// TwinCAT 3 PLC project Untitled2
// Title: Projet Ligne
// Company: Gotec SA
// ProjectVersion: 0.0
// ProgramVersion: 3.1.0.8
// libraries:
//   Recipe Management, 3.4.1.0 (System)
//   Tc2_Standard, * (Beckhoff Automation GmbH)
//   Tc2_System, * (Beckhoff Automation GmbH)
//   Tc3_Interfaces, * (Beckhoff Automation GmbH)
//   Tc3_Module, * (Beckhoff Automation GmbH)
// project tree:
//   / PlcTask.TcTTO
//   POUs/ MAIN.TcPOU
// real-time tasks:
//   TASK PlcTask: cycle T#10ms, priority 20, ADS port 350
// I/O:
//   DEVICE Device 2 (EtherCAT), AmsNetId 10.10.10.31.3.1
//     Grande armoire [EK1100 EtherCAT Coupler (2A E-Bus)]
//       Term 51 (EL1002) [EL1002 2Ch. Dig. Input 24V, 3ms]
//       Term 52 (EL1002) [EL1002 2Ch. Dig. Input 24V, 3ms]
//       Term 53 (EL1002) [EL1002 2Ch. Dig. Input 24V, 3ms]
//       Term 54 (EL1002) [EL1002 2Ch. Dig. Input 24V, 3ms]
//       Term 55 (EL1002) [EL1002 2Ch. Dig. Input 24V, 3ms]
//       Term 56 (EL1002) [EL1002 2Ch. Dig. Input 24V, 3ms]
//       Term 57 (EL1002) [EL1002 2Ch. Dig. Input 24V, 3ms]
//       Term 58 (EL1002) [EL1002 2Ch. Dig. Input 24V, 3ms]
//       Term 59 (EL1002) [EL1002 2Ch. Dig. Input 24V, 3ms]
//       Term 60 (EL1002) [EL1002 2Ch. Dig. Input 24V, 3ms]
//       Term 61 (EL1002) [EL1002 2Ch. Dig. Input 24V, 3ms]
//       Term 62 (EL1002) [EL1002 2Ch. Dig. Input 24V, 3ms]
//       Term 63 (EL1002) [EL1002 2Ch. Dig. Input 24V, 3ms]
//       Term 64 (EL1002) [EL1002 2Ch. Dig. Input 24V, 3ms]
//       Term 65 (EL1002) [EL1002 2Ch. Dig. Input 24V, 3ms]
//       Term 66 (EL1002) [EL1002 2Ch. Dig. Input 24V, 3ms]
//       Term 67 (EL1002) [EL1002 2Ch. Dig. Input 24V, 3ms]
//       Term 68 (EL1002) [EL1002 2Ch. Dig. Input 24V, 3ms]
//       Term 69 (EL1002) [EL1002 2Ch. Dig. Input 24V, 3ms]
//       Term 70 (EL1002) [EL1002 2Ch. Dig. Input 24V, 3ms]
//       Term 71 (EL9410) [EL9410 E-Bus Power Supplier  (Diagnostics)]
//       Term 72 (EL2002) [EL2002 2Ch. Dig. Output 24V, 0.5A]
//       Term 73 (EL2002) [EL2002 2Ch. Dig. Output 24V, 0.5A]
//       Term 74 (EL2002) [EL2002 2Ch. Dig. Output 24V, 0.5A]
//       Term 75 (EL2002) [EL2002 2Ch. Dig. Output 24V, 0.5A]
//       Term 76 (EL2002) [EL2002 2Ch. Dig. Output 24V, 0.5A]
//       Term 77 (EL2002) [EL2002 2Ch. Dig. Output 24V, 0.5A]
//       Term 78 (EL2002) [EL2002 2Ch. Dig. Output 24V, 0.5A]
//       Term 79 (EL2002) [EL2002 2Ch. Dig. Output 24V, 0.5A]
//       Term 80 (EL1512) [EL1512 2Ch. +/- Counter 24V, 1kHz]
//       Term 81 (EL2622) [EL2622 2Ch. Relay Output, NO (230V AC / 30V DC)]
//       Term 82 (EL2622) [EL2622 2Ch. Relay Output, NO (230V AC / 30V DC)]
//       Term 83 (EL2622) [EL2622 2Ch. Relay Output, NO (230V AC / 30V DC)]
//       Term 84 (EL2622) [EL2622 2Ch. Relay Output, NO (230V AC / 30V DC)]
//       Term 85 (EL2622) [EL2622 2Ch. Relay Output, NO (230V AC / 30V DC)]
//       Term 86 (EL2622) [EL2622 2Ch. Relay Output, NO (230V AC / 30V DC)]
//       Term 87 (EL3681) [EL3681 Digital multimeter terminal]
//       Term 88 (EL3681) [EL3681 Digital multimeter terminal]
//       Term 89 (EL6751) [EL6751 CANopen Master]
//       Term 90 (EL6751) [EL6751 CANopen Master]
//       Term 117 (EL9011) [EL9011 End Terminal]
//     Petite armoire [EK1100 EtherCAT Coupler (2A E-Bus)]
//       Term 92 (EL1002) [EL1002 2Ch. Dig. Input 24V, 3ms]
//       Term 93 (EL1002) [EL1002 2Ch. Dig. Input 24V, 3ms]
//       Term 94 (EL1002) [EL1002 2Ch. Dig. Input 24V, 3ms]
//       Term 95 (EL1002) [EL1002 2Ch. Dig. Input 24V, 3ms]
//       Term 96 (EL1002) [EL1002 2Ch. Dig. Input 24V, 3ms]
//       Term 97 (EL1002) [EL1002 2Ch. Dig. Input 24V, 3ms]
//       Term 98 (EL1002) [EL1002 2Ch. Dig. Input 24V, 3ms]
//       Term 99 (EL1002) [EL1002 2Ch. Dig. Input 24V, 3ms]
//       Term 100 (EL1002) [EL1002 2Ch. Dig. Input 24V, 3ms]
//       Term 101 (EL1002) [EL1002 2Ch. Dig. Input 24V, 3ms]
//       Term 102 (EL1002) [EL1002 2Ch. Dig. Input 24V, 3ms]
//       Term 103 (EL1002) [EL1002 2Ch. Dig. Input 24V, 3ms]
//       Term 104 (EL2002) [EL2002 2Ch. Dig. Output 24V, 0.5A]
//       Term 105 (EL2002) [EL2002 2Ch. Dig. Output 24V, 0.5A]
//       Term 106 (EL2002) [EL2002 2Ch. Dig. Output 24V, 0.5A]
//       Term 107 (EL2002) [EL2002 2Ch. Dig. Output 24V, 0.5A]
//       Term 108 (EL3051) [EL3051 1Ch. Ana. Input 4-20mA]
//       Term 109 (EL9512) [EL9512 Power supply terminal 12V]
//       Term 110 (EL3356-0010) [EL3356-0010 1Ch. Ana. Input Resistor Bridge Terminal, 24bit, High Precision]
//       Term 111 (EL9512) [EL9512 Power supply terminal 12V]
//       Term 112 (EL3356-0010) [EL3356-0010 1Ch. Ana. Input Resistor Bridge Terminal, 24bit, High Precision]
//       Term 113 (EL6900) [EL6900, TwinSAFE PLC]
//       Term 114 (EL1904) [EL1904, 4 Ch. Safety Input 24V, TwinSAFE]
//         modules: Module 1 (FSOES)
//       Term 115 (EL1904) [EL1904, 4 Ch. Safety Input 24V, TwinSAFE]
//         modules: Module 1 (FSOES)
//       Term 116 (EL6731) [EL6731 PROFIBUS DP Master]
//       Term 118 (EL9011) [EL9011 End Terminal]
//     Box Etanchetie (EX260-SEC1) [EX260-SEC1 EtherCAT SI Unit (32DO_PNP) Rev1.2]
//     Box Debit (EX260-SEC1) [EX260-SEC1 EtherCAT SI Unit (32DO_PNP) Rev1.2]
//     Box Imprimante (EX260-SEC1) [EX260-SEC1 EtherCAT SI Unit (32DO_PNP) Rev1.2]
//   DEVICE Device 3 (EL6751), AmsNetId 10.10.10.31.4.1
//     Moteur Q1 (EPOS)
//   DEVICE Device 4 (EL6751), AmsNetId 10.10.10.31.5.1
//     Moteur Q2 (EPOS)
//   DEVICE Device 1 (EL6731), AmsNetId 10.10.10.31.2.1
//     Pressure Sensor 2P1 // Vendor: WIKA Revision: Rev 0.2
//     Pressure Sensor 4P2 // Vendor: WIKA Revision: Rev 0.2
//     Pressure Sensor 5P1 // Vendor: WIKA Revision: Rev 0.2
//     Pressure Sensor 5P2 // Vendor: WIKA Revision: Rev 0.2
//     Pressure Sensor 6P1 // Vendor: WIKA Revision: Rev 0.2
//     Pressure Sensor 4P1 // Vendor: WIKA Revision: Rev 0.2

CONFIGURATION Untitled2
    RESOURCE PLC ON TwinCAT3
        TASK PlcTask(INTERVAL := T#10ms, PRIORITY := 20);
        PROGRAM MAIN WITH PlcTask : MAIN;
    END_RESOURCE
END_CONFIGURATION

// ---- POUs/MAIN.TcPOU
PROGRAM MAIN
VAR
END_VAR

END_PROGRAM
